Universal Robots PolyScope program: sync_reach_real.urp

Program test_thread (installation=default directory=/ursim/programs createdIn=3.2.19275 lastSavedIn=5.24.0 robotSerialNumber=20195399999)
Calibrated DH parameters: a=[0, -0.24355, -0.2132, 0, 0, 0]; d=[0.15185, 0, 0, 0.13105, 0.08535, 0.0921]; alpha=[1.570796, 0, 0, 1.570796, -1.570796, 0]; deltaTheta=[0, 0, 0, 0, 0, 0]
InitVariablesNode
BeforeStart
  setp := p[0,0,0,0,0,0]
  Script: rtde_set_watchdog("input_int_register_0", 0.01, "PAUSE")
  Script: write_output_integer_register(0, 1)
  Script: write_output_integer_register(1, 1)
  Script: write_output_integer_register(2, 12345)
Robot Program (runOnlyOnce=false)
  If read_input_integer_register(0)≟1 and setp≠p[0, 0, 0, 0, 0, 0]
    'Valid pose received from client'
    MoveJ speed 60 deg/s, acceleration 80 deg/s^2 (useActiveTCP=true optimoveEnabled=false optiMoveSpeed=0.3 optiMoveAcceleration=0.09) feature=Base
      Waypoint Variable (Variable): variable=setp
    'Confirm that move was executed'
    Script: write_output_integer_register(0, 0)
    'Wait until script acknowledges confirmation'
    Loop While (checkContinuously=false) expression=read_input_integer_register(0)≟1
      Script: sync()
    'Request next pose'
    Script: write_output_integer_register(0, 1)
  Script: sync()
Thread Thread_1 (runOnlyOnce=false)
  Loop Forever
    tmp := p[0,0,0,0,0,0]
    Script: tmp[0] = read_input_float_register(0)
    Script: tmp[1] = read_input_float_register(1)
    Script: tmp[2] = read_input_float_register(2)
    Script: tmp[3] = read_input_float_register(3)
    Script: tmp[4] = read_input_float_register(4)
    Script: tmp[5] = read_input_float_register(5)
    setp := tmp
    Script: sync()
Thread Thread_2 (runOnlyOnce=false)
  prev_req := 0
  Loop Forever
    req := read_input_integer_register(1)
    If req≟1 and prev_req≟0
      tmp2 := p[0,0,0,0,0,0]
      Script: tmp2[0] = read_input_float_register(6)
      Script: tmp2[1] = read_input_float_register(7)
      Script: tmp2[2] = read_input_float_register(8)
      Script: tmp2[3] = read_input_float_register(9)
      Script: tmp2[4] = read_input_float_register(10)
      Script: tmp2[5] = read_input_float_register(11)
      goalp := tmp2
      If get_inverse_kin_has_solution(goalp)
        Script: write_output_integer_register(1, 0)
      Else 
        Script: write_output_integer_register(1, -1)
    If req≟0 and prev_req≟1
      Script: write_output_integer_register(1, 1)
    prev_req := req
    Script: sync()
